// TIA Portal project "BurnerAlarm_Proj" (V17)

(* hardware
DEVICE "PLC_1"  S7-1200 Station
   slot 0: "Rack_0"  S7-1200 Rack  Rack  V1.0
   slot 1: "PLC_1"  CPU 1214C DC/DC/DC  6ES7 214-1AG40-0XB0  V4.5
*)

// ===== PLC "PLC_1"  CPU 1214C DC/DC/DC =====

VAR_GLOBAL   // PLC tag table "烧嘴报警变量"
   "1#故障反馈" AT %I0.1 : Bool;
   "2#故障反馈" AT %I0.4 : Bool;
   "3#故障反馈" AT %I0.7 : Bool;
   "4#故障反馈" AT %I1.2 : Bool;
   "5#故障反馈" AT %I1.5 : Bool;
   "6#故障反馈" AT %I2.2 : Bool;
   "7#故障反馈" AT %I2.5 : Bool;
   "蜂鸣器" AT %Q4.7 : Bool;
END_VAR

DATA_BLOCK "内部数据"   // DB1
{ S7_Optimized_Access := 'TRUE' }
VERSION : 0.1
   VAR
      报警脉冲 : Bool;   // P_TRIG上升沿存储位
      控温超温标志 : Bool;   // 任意区超温标志汇总
   END_VAR
BEGIN
END_DATA_BLOCK

DATA_BLOCK "数字量信号"   // DB2
{ S7_Optimized_Access := 'TRUE' }
VERSION : 0.1
   VAR
      区1超温标志 : Bool;   // 1区超温标志
      区2超温标志 : Bool;   // 2区超温标志
      区3超温标志 : Bool;   // 3区超温标志
      区4超温标志 : Bool;   // 4区超温标志
      区5超温标志 : Bool;   // 5区超温标志
      区6超温标志 : Bool;   // 6区超温标志
   END_VAR
BEGIN
END_DATA_BLOCK

ORGANIZATION_BLOCK "Main"   // OB1, LAD, ProgramCycle
TITLE = "Main Program Sweep (Cycle)"
{ S7_Optimized_Access := 'TRUE' }
VERSION : 0.1
   VAR_INPUT
      Initial_Call : Bool;   // Initial call of this OB
      Remanence : Bool;   // =True, if remanent data are available
   END_VAR
BEGIN
END_ORGANIZATION_BLOCK